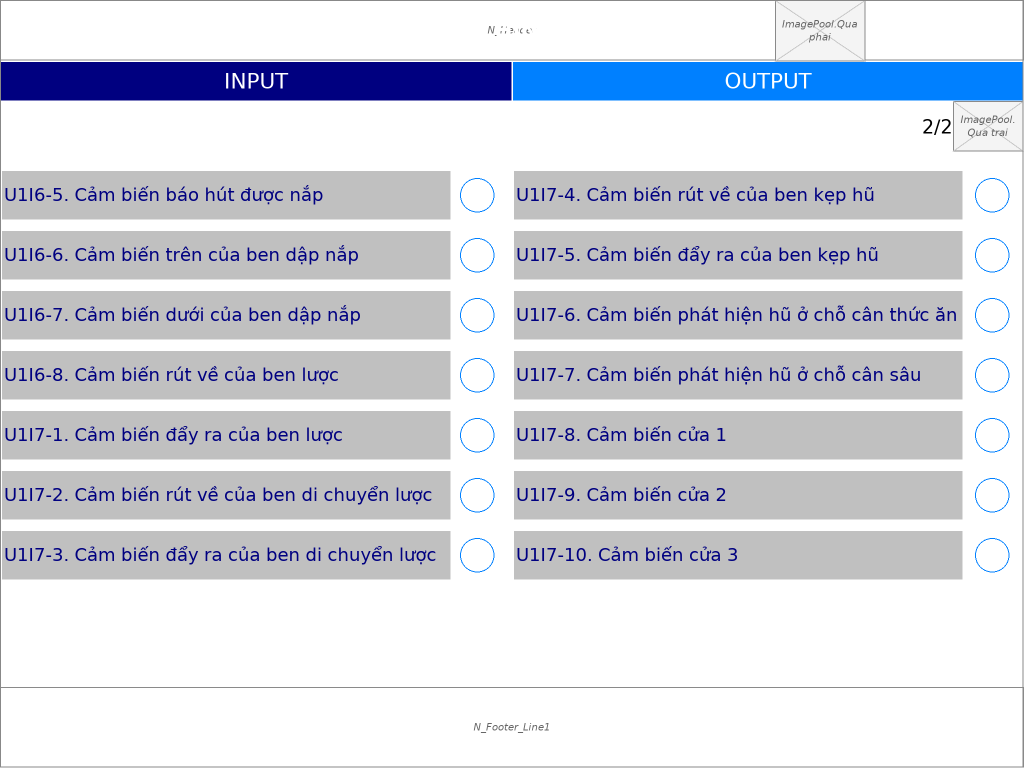
VISUALIZATION N_PLC_I1_next  // 1024x768
    Rectangle (886,102 103x50), "2/2"
    Frame (0,687 1024x80)
        shows N_Footer_Line1()
    Frame (0,0 1024x60)
        shows N_Header()
    Textfield (353,5 400x50), "MÀN HÌNH IO LINE 1"
    Rectangle (0,61 512x40), "INPUT"
        OnMouseClick: change screen: N_PLC_I1
    Rectangle (512,61 512x40), "OUTPUT"
        OnMouseClick: change screen: N_PLC_O1
    Image (775,0 90x61), image: ImagePool.Qua phai
        OnMouseClick: change screen: N_PLC_I2
    Rectangle (1,170 450x50), "U1I6-5. Cảm biến báo hút được nắp"
    Rectangle (1,230 450x50), "U1I6-6. Cảm biến trên của ben dập nắp"
    Rectangle (1,350 450x50), "U1I6-8. Cảm biến rút về của ben lược"
    Rectangle (1,290 450x50), "U1I6-7. Cảm biến dưới của ben dập nắp"
    Rectangle (1,410 450x50), "U1I7-1. Cảm biến đẩy ra của ben lược"
    Rectangle (1,470 450x50), "U1I7-2. Cảm biến rút về của ben di chuyển lược"
    Rectangle (1,530 450x50), "U1I7-3. Cảm biến đẩy ra của ben di chuyển lược"
    Ellipse (460,178 34x34), colour toggle: PR_Line01.fb_LidSupply.fbLidSuctionValve.bPressure, input disabled if: true
    Ellipse (460,238 34x34), colour toggle: PR_Line01.fb_LidClose.fbCylinder_LidClose.bAtRetract, input disabled if: true
    Ellipse (460,298 34x34), colour toggle: PR_Line01.fb_LidClose.fbCylinder_LidClose.bAtExtend, input disabled if: true
    Ellipse (460,358 34x34), colour toggle: PR_Line01.fb_Transfer.fbCylinder_Comb.bAtRetract, input disabled if: true
    Ellipse (460,418 34x34), colour toggle: PR_Line01.fb_Transfer.fbCylinder_Comb.bAtExtend, input disabled if: true
    Ellipse (460,478 34x34), colour toggle: PR_Line01.fb_Transfer.fbCylinder_Move_Comb.bAtRetract, input disabled if: true
    Ellipse (460,538 34x34), colour toggle: PR_Line01.fb_Transfer.fbCylinder_Move_Comb.bAtExtend, input disabled if: true
    Rectangle (513,230 450x50), "U1I7-5. Cảm biến đẩy ra của ben kẹp hũ"
    Rectangle (513,170 450x50), "U1I7-4. Cảm biến rút về của ben kẹp hũ"
    Rectangle (513,290 450x50), "U1I7-6. Cảm biến phát hiện hũ ở chỗ cân thức ăn"
    Rectangle (513,350 450x50), "U1I7-7. Cảm biến phát hiện hũ ở chỗ cân sâu"
    Rectangle (513,410 450x50), "U1I7-8. Cảm biến cửa 1"
    Rectangle (513,470 450x50), "U1I7-9. Cảm biến cửa 2"
    Rectangle (513,530 450x50), "U1I7-10. Cảm biến cửa 3"
    Ellipse (975,178 34x34), colour toggle: PR_Line01.fb_Transfer.fbCylinder_Clip.bAtExtend, input disabled if: true
    Ellipse (975,238 34x34), colour toggle: PR_Line01.fb_Transfer.fbCylinder_Clip.bAtRetract, input disabled if: true
    Ellipse (975,298 34x34), colour toggle: PR_Line01.fb_FoodWeight.bCupPresent, input disabled if: true
    Ellipse (975,358 34x34), colour toggle: PR_Line01.fb_WormWeight.bCupPresent, input disabled if: true
    Ellipse (975,418 34x34), colour toggle: GVL_IO.bSafetyDoor1, input disabled if: true
    Ellipse (975,478 34x34), colour toggle: GVL_IO.bSafetyDoor2, input disabled if: true
    Ellipse (975,538 34x34), colour toggle: GVL_IO.bSafetyDoor3, input disabled if: true
    Image (953,101 70x50), image: ImagePool.Qua trai
        OnMouseClick: change screen: N_PLC_I1
END_VISUALIZATION

(* stored: Version 1.1.0.1, ProductVersion 3.1.4024.12
   Visu N_PLC_I1_next: Id {05c9e358-2f15-452a-b9b4-5eeb3b3ae3cc} *)
